Fanuc KAREL source: compact_preamble.KL

PROGRAM KT00084
%NOLOCKGROUP
VAR
Y1 : ARRAY[2] OF BYTE
R2:REAL
OUT:REAL
BEGIN
Y1[1]=2
R2=3.0
OUT=((Y1[1]) * R2)
END KT00084
